FUNCTION_BLOCK FB_LamparaConmutada_IL
VAR_INPUT
END_VAR
VAR_OUTPUT
END_VAR
VAR
    Lampara AT %Q*: BOOL;
    Pulsador AT %I*: BOOL;
    
    Pulsacion: R_TRIG;
END_VAR

// NETWORK 1
// instruction list
CAL     Pulsacion(
    CLK     := Pulsador)

// NETWORK 2
// instruction list
LD      Pulsacion.Q
JMPCN   End

// NETWORK 3
// instruction list
LDN     Lampara
ST      Lampara

// NETWORK 4
End:
// instruction list

END_FUNCTION_BLOCK

(* stored: Version 1.1.0.1, ProductVersion 3.1.4024.12
   POU FB_LamparaConmutada_IL: Id {4fae365c-fc76-4aae-81b4-957177e5a0b8}, SpecialFunc None *)
